// TIA Portal V19 export
FUNCTION "CollectAlarms" : Void   // FC71, LAD
TITLE = Alarm Collector Unit
// Collects alarms from the respective level and categorises the alarms into the different alarm classes. Filling the alarm DB with specific alarm messages which are defined in the comment of the defined alarm. The definition of possible alarms within a equipment is handled here.
// stored: Namespace Unit2.EM3, SetENOAutomatically false
   VAR_INPUT
      resetAlarms : Bool;
      disableAlarms : Bool;
   END_VAR
   VAR_OUTPUT
      commandsToUnit : "LUC_typeStateCommands";   // Feedback to the unit
   END_VAR
   VAR_TEMP   // added for the SCL form of the ladder/FBD networks
      _w1 : Bool;
   END_VAR
BEGIN

REGION Network 1: Reset Alarms
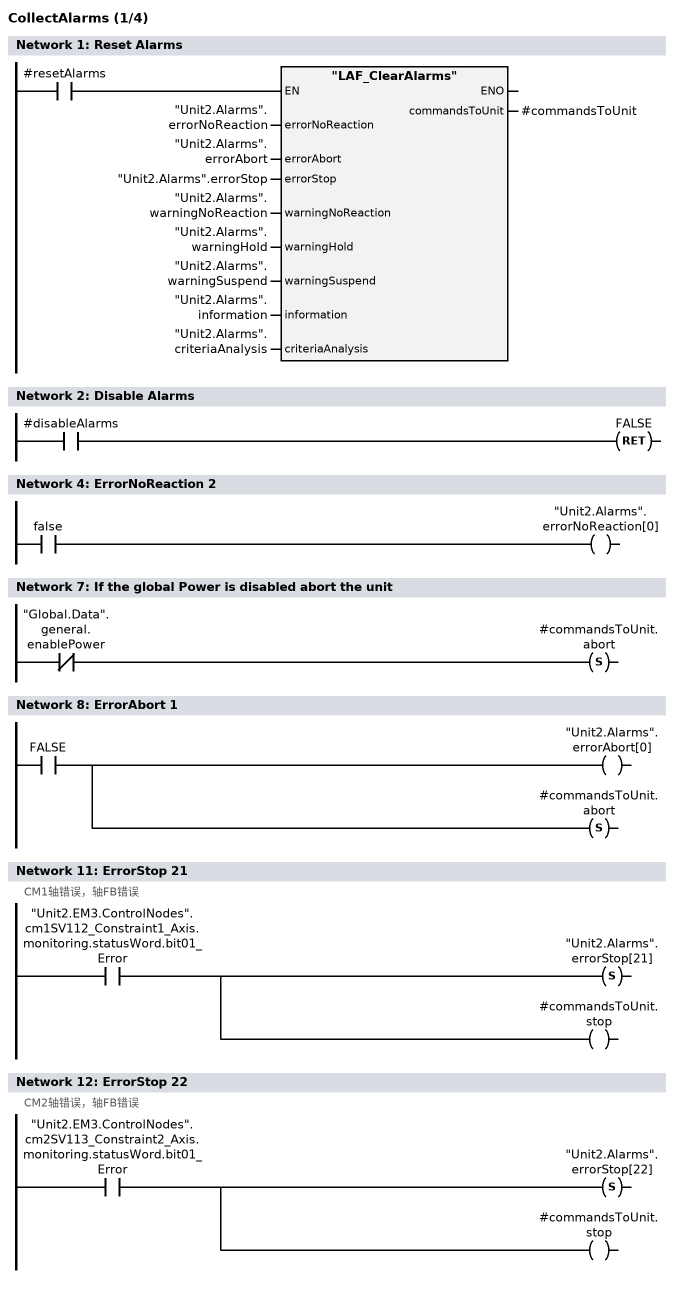
   RUNG wire#powerrail
      Contact( #resetAlarms )
      "LAF_ClearAlarms"(errorNoReaction := "Unit2.Alarms".errorNoReaction, errorAbort := "Unit2.Alarms".errorAbort, errorStop := "Unit2.Alarms".errorStop, warningNoReaction := "Unit2.Alarms".warningNoReaction, warningHold := "Unit2.Alarms".warningHold, warningSuspend := "Unit2.Alarms".warningSuspend, information := "Unit2.Alarms".information, criteriaAnalysis := "Unit2.Alarms".criteriaAnalysis, commandsToUnit => #commandsToUnit)
   END_RUNG
   // the same network as SCL:
   IF #resetAlarms THEN
       "LAF_ClearAlarms"(errorNoReaction := "Unit2.Alarms".errorNoReaction,
                         errorAbort := "Unit2.Alarms".errorAbort,
                         errorStop := "Unit2.Alarms".errorStop,
                         warningNoReaction := "Unit2.Alarms".warningNoReaction,
                         warningHold := "Unit2.Alarms".warningHold,
                         warningSuspend := "Unit2.Alarms".warningSuspend,
                         information := "Unit2.Alarms".information,
                         criteriaAnalysis := "Unit2.Alarms".criteriaAnalysis,
                         commandsToUnit => #commandsToUnit);
   END_IF;
END_REGION

REGION Network 2: Disable Alarms
   RUNG wire#powerrail
      Contact( #disableAlarms )
      ReturnCoil( FALSE )
   END_RUNG
   // the same network as SCL:
   IF #disableAlarms THEN
       ENO := FALSE;
       RETURN;
   END_IF;
END_REGION

REGION Network 3: *************** Error No Reaction ************************
END_REGION

REGION Network 4: ErrorNoReaction 2
   RUNG wire#powerrail
      Contact( false )
      Coil( "Unit2.Alarms".errorNoReaction[0] )
   END_RUNG
   // the same network as SCL:
   "Unit2.Alarms".errorNoReaction[0] := false;
END_REGION

REGION Network 6: *************** Error and Abort **************************
END_REGION

REGION Network 7: If the global Power is disabled abort the unit
   RUNG wire#powerrail
      I_Contact( "Global.Data".general.enablePower )
      S_Coil( #commandsToUnit.abort )
   END_RUNG
   // the same network as SCL:
   IF NOT "Global.Data".general.enablePower THEN #commandsToUnit.abort := TRUE; END_IF;
END_REGION

REGION Network 8: ErrorAbort 1
   RUNG wire#powerrail
      Contact( FALSE )
      wire#w1
      Coil( "Unit2.Alarms".errorAbort[0] )
   END_RUNG
   RUNG wire#w1
      S_Coil( #commandsToUnit.abort )
   END_RUNG
   // the same network as SCL:
   "Unit2.Alarms".errorAbort[0] := FALSE;
   IF FALSE THEN #commandsToUnit.abort := TRUE; END_IF;
END_REGION

REGION Network 10: *************** Error and Stop ***************************
END_REGION

REGION Network 11: ErrorStop 21
   // CM1轴错误，轴FB错误
   RUNG wire#powerrail
      Contact( "Unit2.EM3.ControlNodes".cm1SV112_Constraint1_Axis.monitoring.statusWord.bit01_Error )
      wire#w1
      S_Coil( "Unit2.Alarms".errorStop[21] )
   END_RUNG
   RUNG wire#w1
      Coil( #commandsToUnit.stop )
   END_RUNG
   // the same network as SCL:
   IF "Unit2.EM3.ControlNodes".cm1SV112_Constraint1_Axis.monitoring.statusWord.bit01_Error THEN
       "Unit2.Alarms".errorStop[21] := TRUE;
   END_IF;
   #commandsToUnit.stop := "Unit2.EM3.ControlNodes".cm1SV112_Constraint1_Axis.monitoring.statusWord.bit01_Error;
END_REGION

REGION Network 12: ErrorStop 22
   // CM2轴错误，轴FB错误
   RUNG wire#powerrail
      Contact( "Unit2.EM3.ControlNodes".cm2SV113_Constraint2_Axis.monitoring.statusWord.bit01_Error )
      wire#w1
      S_Coil( "Unit2.Alarms".errorStop[22] )
   END_RUNG
   RUNG wire#w1
      Coil( #commandsToUnit.stop )
   END_RUNG
   // the same network as SCL:
   IF "Unit2.EM3.ControlNodes".cm2SV113_Constraint2_Axis.monitoring.statusWord.bit01_Error THEN
       "Unit2.Alarms".errorStop[22] := TRUE;
   END_IF;
   #commandsToUnit.stop := "Unit2.EM3.ControlNodes".cm2SV113_Constraint2_Axis.monitoring.statusWord.bit01_Error;
END_REGION

REGION Network 13: ErrorStop 23
   // CM3轴错误，轴FB错误
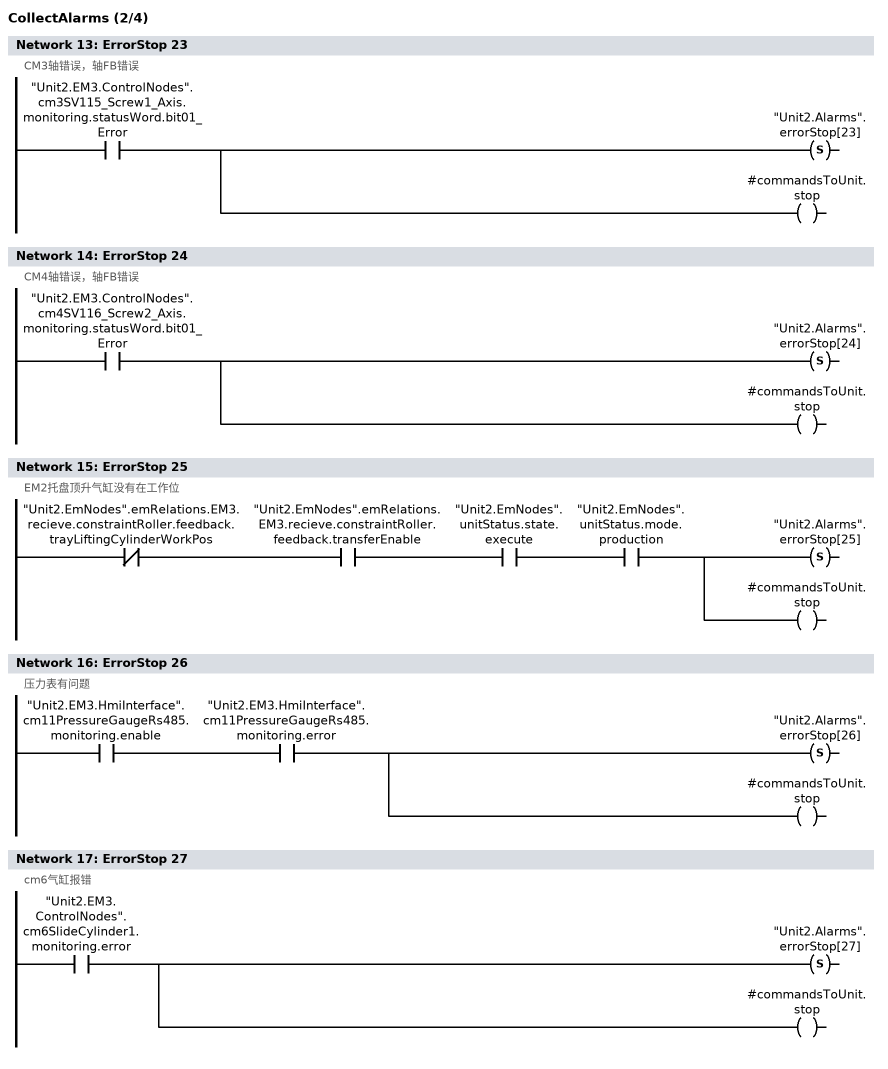
   RUNG wire#powerrail
      Contact( "Unit2.EM3.ControlNodes".cm3SV115_Screw1_Axis.monitoring.statusWord.bit01_Error )
      wire#w1
      S_Coil( "Unit2.Alarms".errorStop[23] )
   END_RUNG
   RUNG wire#w1
      Coil( #commandsToUnit.stop )
   END_RUNG
   // the same network as SCL:
   IF "Unit2.EM3.ControlNodes".cm3SV115_Screw1_Axis.monitoring.statusWord.bit01_Error THEN
       "Unit2.Alarms".errorStop[23] := TRUE;
   END_IF;
   #commandsToUnit.stop := "Unit2.EM3.ControlNodes".cm3SV115_Screw1_Axis.monitoring.statusWord.bit01_Error;
END_REGION

REGION Network 14: ErrorStop 24
   // CM4轴错误，轴FB错误
   RUNG wire#powerrail
      Contact( "Unit2.EM3.ControlNodes".cm4SV116_Screw2_Axis.monitoring.statusWord.bit01_Error )
      wire#w1
      S_Coil( "Unit2.Alarms".errorStop[24] )
   END_RUNG
   RUNG wire#w1
      Coil( #commandsToUnit.stop )
   END_RUNG
   // the same network as SCL:
   IF "Unit2.EM3.ControlNodes".cm4SV116_Screw2_Axis.monitoring.statusWord.bit01_Error THEN
       "Unit2.Alarms".errorStop[24] := TRUE;
   END_IF;
   #commandsToUnit.stop := "Unit2.EM3.ControlNodes".cm4SV116_Screw2_Axis.monitoring.statusWord.bit01_Error;
END_REGION

REGION Network 15: ErrorStop 25
   // EM2托盘顶升气缸没有在工作位
   RUNG wire#powerrail
      I_Contact( "Unit2.EmNodes".emRelations.EM3.recieve.constraintRoller.feedback.trayLiftingCylinderWorkPos )
      Contact( "Unit2.EmNodes".emRelations.EM3.recieve.constraintRoller.feedback.transferEnable )
      Contact( "Unit2.EmNodes".unitStatus.state.execute )
      Contact( "Unit2.EmNodes".unitStatus.mode.production )
      wire#w1
      S_Coil( "Unit2.Alarms".errorStop[25] )
   END_RUNG
   RUNG wire#w1
      Coil( #commandsToUnit.stop )
   END_RUNG
   // the same network as SCL:
   #_w1 := NOT "Unit2.EmNodes".emRelations.EM3.recieve.constraintRoller.feedback.trayLiftingCylinderWorkPos AND "Unit2.EmNodes".emRelations.EM3.recieve.constraintRoller.feedback.transferEnable AND "Unit2.EmNodes".unitStatus.state.execute AND "Unit2.EmNodes".unitStatus.mode.production;
   IF #_w1 THEN "Unit2.Alarms".errorStop[25] := TRUE; END_IF;
   #commandsToUnit.stop := #_w1;
END_REGION

REGION Network 16: ErrorStop 26
   // 压力表有问题
   RUNG wire#powerrail
      Contact( "Unit2.EM3.HmiInterface".cm11PressureGaugeRs485.monitoring.enable )
      Contact( "Unit2.EM3.HmiInterface".cm11PressureGaugeRs485.monitoring.error )
      wire#w1
      S_Coil( "Unit2.Alarms".errorStop[26] )
   END_RUNG
   RUNG wire#w1
      Coil( #commandsToUnit.stop )
   END_RUNG
   // the same network as SCL:
   #_w1 := "Unit2.EM3.HmiInterface".cm11PressureGaugeRs485.monitoring.enable AND "Unit2.EM3.HmiInterface".cm11PressureGaugeRs485.monitoring.error;
   IF #_w1 THEN "Unit2.Alarms".errorStop[26] := TRUE; END_IF;
   #commandsToUnit.stop := #_w1;
END_REGION

REGION Network 17: ErrorStop 27
   // cm6气缸报错
   RUNG wire#powerrail
      Contact( "Unit2.EM3.ControlNodes".cm6SlideCylinder1.monitoring.error )
      wire#w1
      S_Coil( "Unit2.Alarms".errorStop[27] )
   END_RUNG
   RUNG wire#w1
      Coil( #commandsToUnit.stop )
   END_RUNG
   // the same network as SCL:
   IF "Unit2.EM3.ControlNodes".cm6SlideCylinder1.monitoring.error THEN
       "Unit2.Alarms".errorStop[27] := TRUE;
   END_IF;
   #commandsToUnit.stop := "Unit2.EM3.ControlNodes".cm6SlideCylinder1.monitoring.error;
END_REGION

REGION Network 18: ErrorStop 28
   // cm7气缸报错
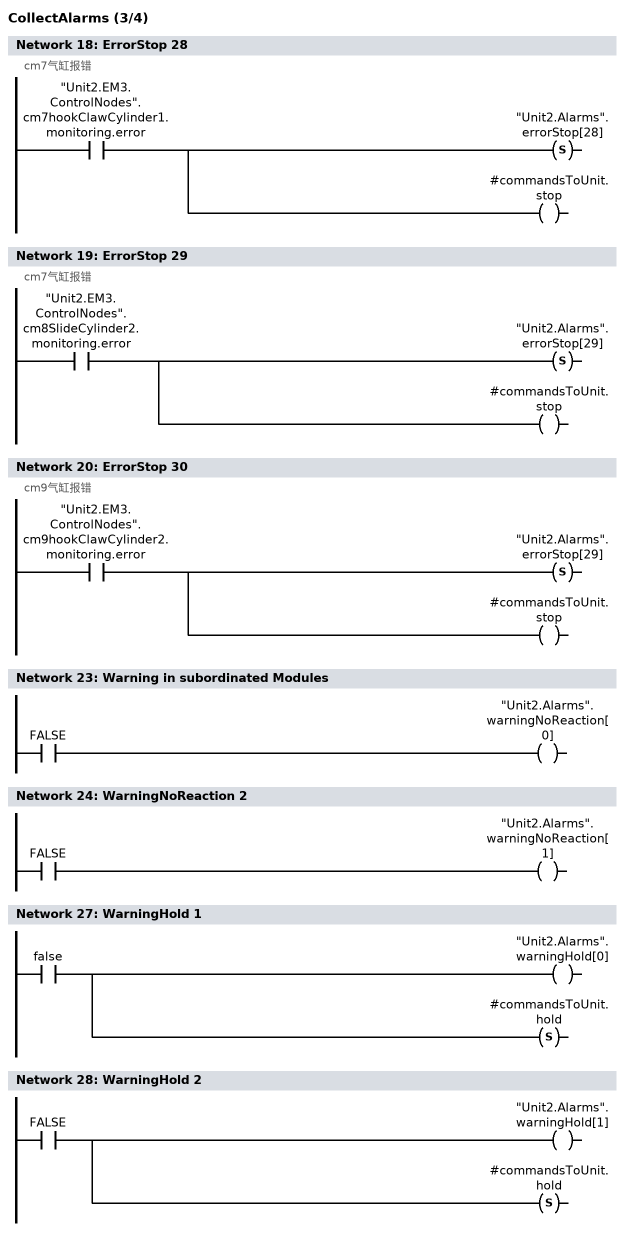
   RUNG wire#powerrail
      Contact( "Unit2.EM3.ControlNodes".cm7hookClawCylinder1.monitoring.error )
      wire#w1
      S_Coil( "Unit2.Alarms".errorStop[28] )
   END_RUNG
   RUNG wire#w1
      Coil( #commandsToUnit.stop )
   END_RUNG
   // the same network as SCL:
   IF "Unit2.EM3.ControlNodes".cm7hookClawCylinder1.monitoring.error THEN
       "Unit2.Alarms".errorStop[28] := TRUE;
   END_IF;
   #commandsToUnit.stop := "Unit2.EM3.ControlNodes".cm7hookClawCylinder1.monitoring.error;
END_REGION

REGION Network 19: ErrorStop 29
   // cm7气缸报错
   RUNG wire#powerrail
      Contact( "Unit2.EM3.ControlNodes".cm8SlideCylinder2.monitoring.error )
      wire#w1
      S_Coil( "Unit2.Alarms".errorStop[29] )
   END_RUNG
   RUNG wire#w1
      Coil( #commandsToUnit.stop )
   END_RUNG
   // the same network as SCL:
   IF "Unit2.EM3.ControlNodes".cm8SlideCylinder2.monitoring.error THEN
       "Unit2.Alarms".errorStop[29] := TRUE;
   END_IF;
   #commandsToUnit.stop := "Unit2.EM3.ControlNodes".cm8SlideCylinder2.monitoring.error;
END_REGION

REGION Network 20: ErrorStop 30
   // cm9气缸报错
   RUNG wire#powerrail
      Contact( "Unit2.EM3.ControlNodes".cm9hookClawCylinder2.monitoring.error )
      wire#w1
      S_Coil( "Unit2.Alarms".errorStop[29] )
   END_RUNG
   RUNG wire#w1
      Coil( #commandsToUnit.stop )
   END_RUNG
   // the same network as SCL:
   IF "Unit2.EM3.ControlNodes".cm9hookClawCylinder2.monitoring.error THEN
       "Unit2.Alarms".errorStop[29] := TRUE;
   END_IF;
   #commandsToUnit.stop := "Unit2.EM3.ControlNodes".cm9hookClawCylinder2.monitoring.error;
END_REGION

REGION Network 22: *************** Warning No Reaction **********************
END_REGION

REGION Network 23: Warning in subordinated Modules
   RUNG wire#powerrail
      Contact( FALSE )
      Coil( "Unit2.Alarms".warningNoReaction[0] )
   END_RUNG
   // the same network as SCL:
   "Unit2.Alarms".warningNoReaction[0] := FALSE;
END_REGION

REGION Network 24: WarningNoReaction 2
   RUNG wire#powerrail
      Contact( FALSE )
      Coil( "Unit2.Alarms".warningNoReaction[1] )
   END_RUNG
   // the same network as SCL:
   "Unit2.Alarms".warningNoReaction[1] := FALSE;
END_REGION

REGION Network 26: *************** Warning Hold **************************
END_REGION

REGION Network 27: WarningHold 1
   RUNG wire#powerrail
      Contact( false )
      wire#w1
      Coil( "Unit2.Alarms".warningHold[0] )
   END_RUNG
   RUNG wire#w1
      S_Coil( #commandsToUnit.hold )
   END_RUNG
   // the same network as SCL:
   "Unit2.Alarms".warningHold[0] := false;
   IF false THEN #commandsToUnit.hold := TRUE; END_IF;
END_REGION

REGION Network 28: WarningHold 2
   RUNG wire#powerrail
      Contact( FALSE )
      wire#w1
      Coil( "Unit2.Alarms".warningHold[1] )
   END_RUNG
   RUNG wire#w1
      S_Coil( #commandsToUnit.hold )
   END_RUNG
   // the same network as SCL:
   "Unit2.Alarms".warningHold[1] := FALSE;
   IF FALSE THEN #commandsToUnit.hold := TRUE; END_IF;
END_REGION

REGION Network 30: *************** Warning Suspend ***********************
END_REGION

REGION Network 31: WarningSuspend 1
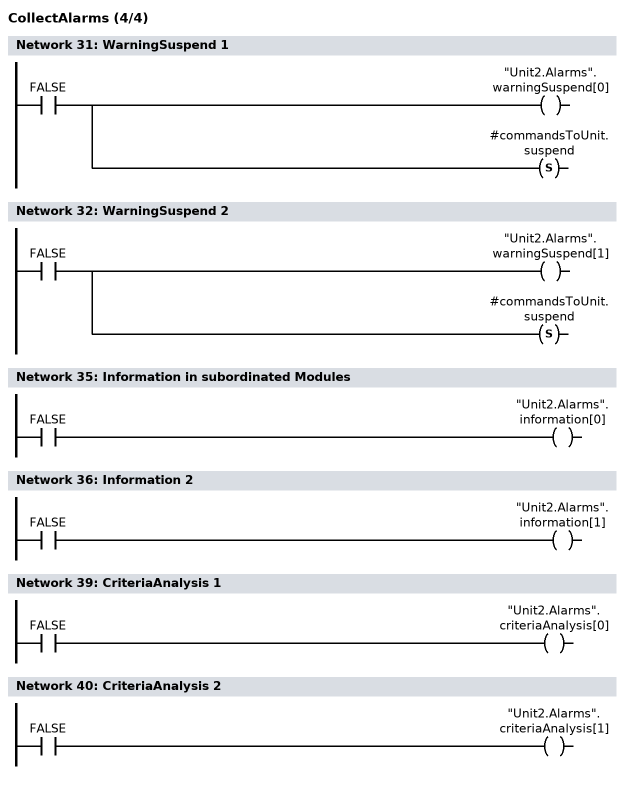
   RUNG wire#powerrail
      Contact( FALSE )
      wire#w1
      Coil( "Unit2.Alarms".warningSuspend[0] )
   END_RUNG
   RUNG wire#w1
      S_Coil( #commandsToUnit.suspend )
   END_RUNG
   // the same network as SCL:
   "Unit2.Alarms".warningSuspend[0] := FALSE;
   IF FALSE THEN #commandsToUnit.suspend := TRUE; END_IF;
END_REGION

REGION Network 32: WarningSuspend 2
   RUNG wire#powerrail
      Contact( FALSE )
      wire#w1
      Coil( "Unit2.Alarms".warningSuspend[1] )
   END_RUNG
   RUNG wire#w1
      S_Coil( #commandsToUnit.suspend )
   END_RUNG
   // the same network as SCL:
   "Unit2.Alarms".warningSuspend[1] := FALSE;
   IF FALSE THEN #commandsToUnit.suspend := TRUE; END_IF;
END_REGION

REGION Network 34: *************** Information *****************************
END_REGION

REGION Network 35: Information in subordinated Modules
   RUNG wire#powerrail
      Contact( FALSE )
      Coil( "Unit2.Alarms".information[0] )
   END_RUNG
   // the same network as SCL:
   "Unit2.Alarms".information[0] := FALSE;
END_REGION

REGION Network 36: Information 2
   RUNG wire#powerrail
      Contact( FALSE )
      Coil( "Unit2.Alarms".information[1] )
   END_RUNG
   // the same network as SCL:
   "Unit2.Alarms".information[1] := FALSE;
END_REGION

REGION Network 38: *************** CriteriaAnalysis **************************
END_REGION

REGION Network 39: CriteriaAnalysis 1
   RUNG wire#powerrail
      Contact( FALSE )
      Coil( "Unit2.Alarms".criteriaAnalysis[0] )
   END_RUNG
   // the same network as SCL:
   "Unit2.Alarms".criteriaAnalysis[0] := FALSE;
END_REGION

REGION Network 40: CriteriaAnalysis 2
   RUNG wire#powerrail
      Contact( FALSE )
      Coil( "Unit2.Alarms".criteriaAnalysis[1] )
   END_RUNG
   // the same network as SCL:
   "Unit2.Alarms".criteriaAnalysis[1] := FALSE;
END_REGION
END_FUNCTION
